// Mitsubishi GX Works2 project: 240528_링카운터조작패널   PLC: Q03UDV

PROGRAM MAIN
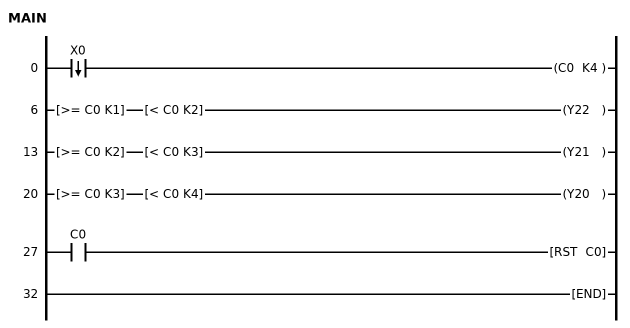
0     LDF     X0
      OUT     C0 K4
6     LD>=    C0 K1
      AND<    C0 K2
      OUT     Y22
13    LD>=    C0 K2
      AND<    C0 K3
      OUT     Y21
20    LD>=    C0 K3
      AND<    C0 K4
      OUT     Y20
27    LD      C0
      RST     C0
32    END
END_PROGRAM
